# EPICS autosave request: iocs/zmqIOC/iocBoot/iocZMQ/auto_settings.req
file "ADBase_settings.req",         P=$(P),  R=cam1:
file "NDPluginBase_settings.req",   P=$(P),  R=image1:
file "NDStdArrays_settings.req",    P=$(P),  R=image1:
file "ADZMQ_settings.req",          P=$(P),  R=ZMQ1:
file "commonPlugin_settings.req",   P=$(P)
